FUNCTION_BLOCK FB_PipelineStage
VAR_INPUT
    value : INT;
END_VAR
VAR_OUTPUT
    bError : BOOL;
END_VAR
VAR
    inner : FB_PipelineInner;
END_VAR

METHOD Step : INT
inner(value := value);
// MISSING: bError := inner.bError;
Step := value;
END_METHOD

END_FUNCTION_BLOCK

(* stored: Version 1.1.0.1
   POU FB_PipelineStage: Id {1918ee7b-13f4-4bcd-8466-37cca1c6c7db}, SpecialFunc None
   Method Step: Id {d0c937b3-f656-4aa9-8ca9-c22da5eef8c9} *)
